RoboDK station: RoboDK Project.rdk

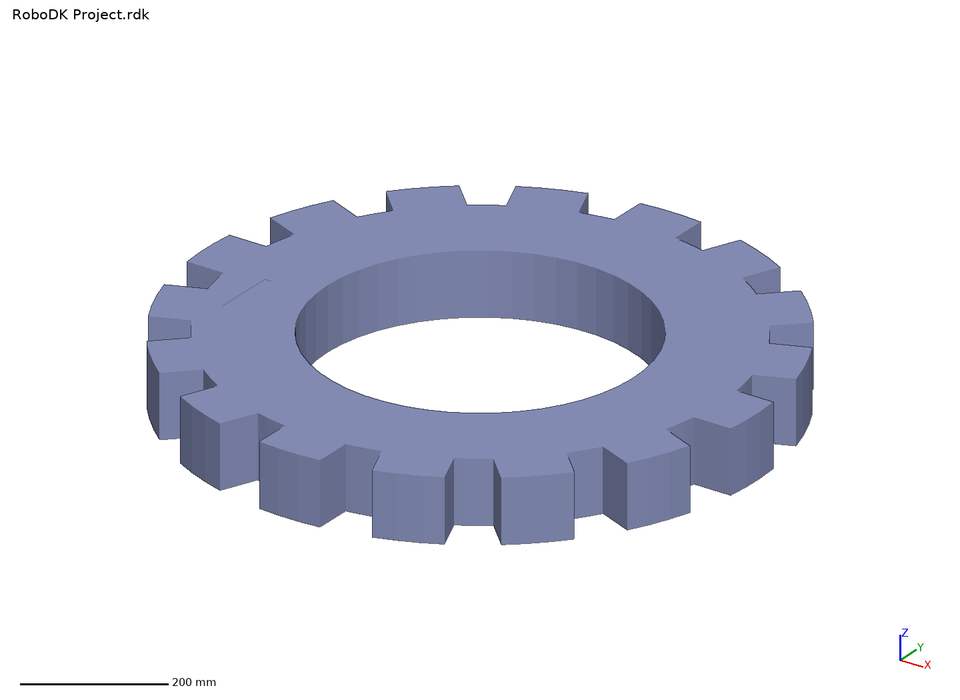
[picture v0: the station drawn from its stored meshes, robots at their saved joint values, targets as dots, program paths as lines]
Station RoboDK Project (saved by RoboDK 5.9.4). Poses are relative to the parent item; angles as X-Y-Z fixed-axis rotations.
Station parameters (name, value as stored): WASM
  - object gear_scratch_master at (0, 0, 0) mm, size 899.4 x 899.4 x 100 mm
